{attribute 'GeneratedUsingTerminal: CU1123-0000-0016'}
{attribute addProperty BoxType "CU1123-0000-0016"}
{attribute addProperty Description "CU1123 EtherCAT junction (3-ports)"}
{attribute addProperty Physics "Y_YY"}
{attribute addProperty Id "InfoDataAT %I*InfoData_6F19DB2B2"}
{attribute addProperty CRC "532711307"}
{attribute addProperty Size "2"}
TYPE CU1123_1FC0878B EXTENDS EtcSlaveBoxBase_77A0E4A7 :
STRUCT
	{attribute addProperty Name "InfoData"}
	InfoData : InfoData_6F19DB2B;
END_STRUCT
END_TYPE

(* stored: Version 1.2.0.0, ProductVersion 3.1.4024.11
   DUT CU1123_1FC0878B: Id {a462461e-450a-44b2-bd02-ace72a9a1725} *)
